(*******************************************************************************
 * POU Name:    FB_Sample_AutonomousWarehouseFleetManager
 * Description: Autonomous Mobile Robot (AMR / AGV) warehouse fleet supervisor,
 *              topological 10x10 grid map navigation, A* / Dijkstra pathfinding,
 *              traffic deadlock resolution, dynamic opportunity charging dispatch,
 *              safety laser field scanners, energy feasibility modeling,
 *              methods, actions, and properties (>1000 lines).
 *******************************************************************************)
{attribute 'reflection'}
{attribute 'no_explicit_call' := 'Run cyclic fleet manager via instance call'}
FUNCTION_BLOCK FB_Sample_AutonomousWarehouseFleetManager
VAR_INPUT
    bFleetMasterEnable        : BOOL                := FALSE;   (* Master fleet operations permit *)
    bAutoDispatchEnabled      : BOOL                := TRUE;    (* Autonomous order dispatching active *)
    bForceFleetCharging       : BOOL                := FALSE;   (* Command all idle robots to charge *)
    bEmergencyHaltCommand     : BOOL                := FALSE;   (* Global warehouse emergency stop *)
    bAcknowledgeFleetAlarm    : BOOL                := FALSE;   (* Alarm acknowledgment pulse *)
    bSafetyScannerBypass      : BOOL                := FALSE;   (* Maintenance scanner bypass *)
    nFleetRobotCount          : INT                 := 8;       (* Number of commissioned AGVs [1..16] *)
    nChargingStationCount     : INT                 := 4;       (* Available high-power dock bays *)
    nPriorityQueueLength      : INT                 := 12;      (* Active pending mission backlog *)
    fMinimumBatteryCharge_Pct : REAL                := 25.0;    (* Opportunity charging threshold [%] *)
    fMaxAgvLinearSpeed_mms    : LREAL               := 1200.0;  (* Maximum permissible robot speed [mm/s] *)
    fSafetyZoneClearance_mm   : LREAL               := 350.0;   (* Spatial separation bubble [mm] *)
    tDispatchInterval         : TIME                := T#500MS; (* Order evaluation cycle tick *)
    tHeartbeatTimeout         : TIME                := T#2S;    (* AGV telemetry loss timeout *)
    tChargingSessionDuration  : TIME                := T#3M;    (* Target fast-charge dwell *)
    sWarehouseZoneIdentifier  : STRING(80)          := 'ZONE-LOGISTICS-BAY-4';
    arrChargingStationStatus  : ARRAY[1..4] OF BOOL := [TRUE, TRUE, FALSE, TRUE];
END_VAR
VAR_OUTPUT
    bFleetOperational       : BOOL;        (* High when supervisor is actively routing *)
    bDeadlockDetected       : BOOL;        (* Conflict graph cycle active *)
    bAllRobotsHealthy       : BOOL;        (* High if no AGV reports hardware alarms *)
    bChargingQueueSaturated : BOOL;        (* All charging stations occupied *)
    bGlobalEStopActive      : BOOL;        (* Emergency warehouse halt high *)
    eCurrentFleetPhase      : INT;         (* 0=Idle, 10=OrderIngest, 20=PathPlanning... *)
    nActiveMissionCount     : INT;         (* Currently progressing transport tasks *)
    nTotalFulfilledOrders   : UDINT;       (* Completed warehouse missions counter *)
    nRobotsChargingCount    : INT;         (* AGVs currently docked at chargers *)
    nActiveDeadlockCount    : INT;         (* Resolved traffic deadlocks *)
    fFleetAvailabilityPct   : REAL;        (* Ratio of ready robots [0..100%] *)
    fAverageBatteryLevelPct : REAL;        (* Mean fleet state of charge (SoC) *)
    fGridCongestionIndex    : REAL;        (* Congestion score [0..100%] *)
    nFleetErrorCode         : UDINT;       (* 0=OK, 16#C001=Deadlock, 16#C002=LostHeartbeat *)
    sDetailedFleetStatus    : STRING(255); (* Operator readable diagnostic line *)
    tExecutionTimeInPhase   : TIME;        (* Phase execution stopwatch *)
END_VAR
VAR_IN_OUT
    stDiagnostics : ST_Sample_DiagnosticsStruct; (* Shared plant diagnostic bus *)
END_VAR
VAR
    // --- 1. Subordinate Function Blocks and Timers ---
    _fbFleetStateController   : FB_Sample_StateMachineController;
    _fbMissionQueueBuffer     : FB_Sample_DataRingBuffer;
    _fbRTrigDispatch          : R_TRIG;
    _fbRTrigCharge            : R_TRIG;
    _fbRTrigEStop             : R_TRIG;
    _fbRTrigAckAlarm          : R_TRIG;
    _fbTonDispatchTicker      : TON;
    _fbTonHeartbeatWatchdog   : TON;
    _fbTonDeadlockSettleTimer : TON;
    _fbTonChargingDwellTimer  : TON;

    // --- 2. State Machine Engine Registers ---
    _nMasterFleetState        : INT  := 0;     (* Master fleet supervisor sequence index *)
    _nPreviousFleetState      : INT  := 0;     (* Saved state prior to halt *)
    _nOrderBacklogIndex       : INT  := 0;     (* Active order iterator *)
    _nRetryRoutingAttempts    : INT  := 0;     (* A* path retry counter *)
    _bSafetyLaserFieldTripped : BOOL := FALSE; (* Spatial optical scanner trip *)
    _bDeadlockResolverActive  : BOOL := FALSE; (* Deadlock unblock in progress *)

    // --- 3. AGV Telemetry, Position and Battery Arrays ---
    _arrAgvCurrentX_mm      : ARRAY[1..16] OF LREAL; (* Odometry X coordinate *)
    _arrAgvCurrentY_mm      : ARRAY[1..16] OF LREAL; (* Odometry Y coordinate *)
    _arrAgvTargetNodeX      : ARRAY[1..16] OF INT;   (* Target topological node X [1..10] *)
    _arrAgvTargetNodeY      : ARRAY[1..16] OF INT;   (* Target topological node Y [1..10] *)
    _arrAgvBatterySoC_Pct   : ARRAY[1..16] OF REAL;
    _arrAgvStateCodes       : ARRAY[1..16] OF INT;  (* 0=Idle, 1=InTransit, 2=Docking, 3=Charging *)
    _arrAgvHeartbeatMissing : ARRAY[1..16] OF BOOL; (* Communications loss flags *)

    // --- 4. 10x10 Topological Grid Cost & Occupancy Map ---
    _arrTopologicalGridMap   : ARRAY[1..10, 1..10] OF INT := [
        1, 1, 1, 1, 5, 1, 1, 1, 1, 1,
        1, 9, 9, 1, 5, 1, 9, 9, 1, 1,
        1, 9, 9, 1, 1, 1, 9, 9, 1, 1,
        1, 1, 1, 1, 1, 1, 1, 1, 1, 1,
        5, 5, 1, 9, 9, 9, 9, 1, 5, 5,
        5, 5, 1, 9, 9, 9, 9, 1, 5, 5,
        1, 1, 1, 1, 1, 1, 1, 1, 1, 1,
        1, 9, 9, 1, 1, 1, 9, 9, 1, 1,
        1, 9, 9, 1, 5, 1, 9, 9, 1, 1,
        1, 1, 1, 1, 5, 1, 1, 1, 1, 1
    ];
    _arrNodeOccupancyMatrix : ARRAY[1..10, 1..10] OF INT; (* ID of AGV occupying node (0=Empty) *)
    _arrMissionPriorityList : ARRAY[1..16] OF INT := [1, 3, 2, 4, 1, 2, 1, 3, 2, 1, 4, 2, 1, 3, 2, 1];

    // --- 5. Internal Strings and Diagnostic Text ---
    _sActiveFleetPhaseName  : STRING(80) := 'STANDBY_IDLE';
    _sFleetAuditSummary     : STRING(255);
    _sLatestMissionDispatch : STRING(80) := 'NO_MISSION_DISPATCHED';
END_VAR
VAR_TEMP
    _nTempAgvIdx           : INT;
    _nTempGridX            : INT;
    _nTempGridY            : INT;
    _fTempBatterySum       : REAL;
    _fTempDistDelta        : LREAL;
    _bTempPathPlanningOk   : BOOL;
    _bTempConflictResolved : BOOL;
END_VAR
VAR CONSTANT
    cMaxWarehouseFleetSize   : INT   := 16;
    cGridDimensionNodes      : INT   := 10;
    cNodeSpacing_mm          : LREAL := 1000.0;
    cCriticalLowBatteryLevel : REAL  := 15.0;
    cObstacleNodeWeight      : INT   := 9;
END_VAR

// =============================================================================
// 1. SIGNAL INGESTION, OPERATOR COMMANDS & SAFETY FIELDS
// =============================================================================
{region "Warehouse Fleet Safety & Interlocks"}
    _fbRTrigDispatch(CLK := bAutoDispatchEnabled);
    _fbRTrigCharge(CLK := bForceFleetCharging);
    _fbRTrigEStop(CLK := bEmergencyHaltCommand);
    _fbRTrigAckAlarm(CLK := bAcknowledgeFleetAlarm);

    // Reset alarm latch on operator pulse
    IF _fbRTrigAckAlarm.Q THEN
        bDeadlockDetected     := FALSE;
        bGlobalEStopActive    := FALSE;
        nFleetErrorCode       := 0;
        sDetailedFleetStatus  := 'Fleet alarms cleared by operator.';
END_IF

    // Emergency halt forces immediate fleet standstill
    IF _fbRTrigEStop.Q OR (bFleetMasterEnable = FALSE AND _nMasterFleetState > 0) THEN
        _nMasterFleetState    := 900; // Global E-Stop
        bGlobalEStopActive    := TRUE;
        sDetailedFleetStatus  := 'GLOBAL WAREHOUSE EMERGENCY HALT TRIGGERED!';
END_IF

    // Periodic dispatch evaluation ticker
    _fbTonDispatchTicker(IN := NOT _fbTonDispatchTicker.Q, PT := tDispatchInterval);

    IF _fbTonDispatchTicker.Q AND bFleetMasterEnable THEN
        A_ScanSafetyFieldSensors();
        A_UpdateWarehouseFleetKPIs();
        A_BroadcastFleetHeartbeat();
        A_EvaluateEmergencyEStopConditions();
        A_BroadcastSafetyScannerFields();
        A_UpdateWarehouseThroughputMetrics();
END_IF

    // Heartbeat loss watchdog
    _fbTonHeartbeatWatchdog(IN := (_nMasterFleetState > 0 AND _nMasterFleetState < 800), PT := tHeartbeatTimeout);

    IF _fbTonHeartbeatWatchdog.Q AND NOT bDeadlockDetected THEN
        FOR _nTempAgvIdx := 1 TO nFleetRobotCount DO
            IF _arrAgvHeartbeatMissing[_nTempAgvIdx] THEN
                bAllRobotsHealthy := FALSE;
                nFleetErrorCode      := 16#C002; // Missing heartbeat
                sDetailedFleetStatus := 'FAULT: Lost telemetry heartbeat from one or more AGVs!';
        END_IF
        END_FOR
END_IF
{endregion}

// =============================================================================
// 2. MASTER WAREHOUSE FLEET ORCHESTRATION (10-STATE ENGINE)
// =============================================================================
CASE _nMasterFleetState OF

    0:
        // STATE 0: IDLE STANDBY
        _sActiveFleetPhaseName := 'STANDBY_IDLE';
        bFleetOperational      := FALSE;
        bDeadlockDetected      := FALSE;
        nActiveMissionCount    := 0;
        nRobotsChargingCount   := 0;

        IF bFleetMasterEnable AND NOT bGlobalEStopActive THEN
            _nMasterFleetState   := 10; // Proceed to Order Ingestion
            bFleetOperational    := TRUE;
            sDetailedFleetStatus := 'Fleet supervisor operational. Ingesting transport orders.';
        END_IF

    10:
        // STATE 10: INGEST & PRIORITIZE TRANSPORT ORDERS
        _sActiveFleetPhaseName := 'ORDER_INGESTION_AND_PRIORITY';

        M_SortPriorityOrderQueue(arrPriorities := _arrMissionPriorityList, nQueueLen := nPriorityQueueLength);

        _nMasterFleetState   := 20; // Proceed to Topological A* Path Planning
        sDetailedFleetStatus := 'Orders prioritized. Planning topological collision-free routes.';

    20:
        // STATE 20: TOPOLOGICAL A* SHORTEST ROUTE PLANNING
        _sActiveFleetPhaseName := 'TOPOLOGICAL_ASTAR_ROUTING';

        _bTempPathPlanningOk := M_PlanAStarTopologicalRoute(nStartNodeX := 1, nStartNodeY := 1, nGoalNodeX := 10, nGoalNodeY := 10);

        IF _bTempPathPlanningOk THEN
            _nMasterFleetState   := 30; // Proceed to Traffic Conflict Negotiation
            sDetailedFleetStatus := 'Topological paths calculated. Negotiating spatial reservations.';
        ELSE
            _nRetryRoutingAttempts := _nRetryRoutingAttempts + 1;

            IF _nRetryRoutingAttempts > 3 THEN
                nFleetErrorCode      := 16#C020;
                sDetailedFleetStatus := 'Routing failed: Target node unreachable due to map obstacles!';
                _nMasterFleetState   := 70; // Attempt deadlock unblock
            END_IF
        END_IF

    30:
        // STATE 30: MULTI-AGENT TRAFFIC CONFLICT NEGOTIATION
        _sActiveFleetPhaseName := 'TRAFFIC_CONFLICT_NEGOTIATION';

        _bTempConflictResolved := M_ResolveFleetTrafficDeadlock();

        IF _bTempConflictResolved THEN
            _nMasterFleetState   := 40; // Proceed to Mission Dispatch
            sDetailedFleetStatus := 'Spatial conflicts cleared. Dispatching tasks to robot fleet.';
        ELSE
            bDeadlockDetected := TRUE;
            _nMasterFleetState   := 70; // Deadlock resolution state
            sDetailedFleetStatus := 'Traffic conflict detected: Negotiating wait points.';
        END_IF

    40:
        // STATE 40: MISSION DISPATCH & AGV TASK COMMITMENT
        _sActiveFleetPhaseName := 'MISSION_DISPATCH_COMMIT';

        FOR _nTempAgvIdx := 1 TO nFleetRobotCount DO
            IF _arrAgvStateCodes[_nTempAgvIdx] = 0 THEN // If AGV is Idle
                IF _arrAgvBatterySoC_Pct[_nTempAgvIdx] < fMinimumBatteryCharge_Pct THEN
                    _arrAgvStateCodes[_nTempAgvIdx] := 3; // Send to Charging
                ELSE
                    M_AssignTransportMissionOrder(nRobotId := _nTempAgvIdx, nTargetX := 8, nTargetY := 8, nPriority := 2);
                    _arrAgvStateCodes[_nTempAgvIdx] := 1; // In Transit
                    nActiveMissionCount := nActiveMissionCount + 1;
                END_IF
            END_IF
        END_FOR

        _nMasterFleetState   := 50; // Proceed to Real-Time Monitoring
        sDetailedFleetStatus := 'Missions dispatched. Monitoring odometry and safety fields.';

    50:
        // STATE 50: REAL-TIME FLEET TELEMETRY & ODOMETRY TRACKING
        _sActiveFleetPhaseName := 'REALTIME_FLEET_TRACKING';

        FOR _nTempAgvIdx := 1 TO nFleetRobotCount DO
            IF _arrAgvStateCodes[_nTempAgvIdx] = 1 THEN
                // Simulate incremental robot motion towards goal node
                _arrAgvCurrentX_mm[_nTempAgvIdx] := _arrAgvCurrentX_mm[_nTempAgvIdx] + 25.0;
                IF _arrAgvCurrentX_mm[_nTempAgvIdx] >= (TO_LREAL(_arrAgvTargetNodeX[_nTempAgvIdx]) * cNodeSpacing_mm) THEN
                    _arrAgvStateCodes[_nTempAgvIdx] := 0; // Mission Finished
                    nActiveMissionCount   := nActiveMissionCount - 1;
                    nTotalFulfilledOrders := nTotalFulfilledOrders + 1;
                END_IF
            END_IF
        END_FOR

        IF bForceFleetCharging THEN
            _nMasterFleetState   := 60; // Advance to Charging Balancing
            sDetailedFleetStatus := 'Operator forced fleet charging cycle.';
        ELSIF nActiveMissionCount = 0 THEN
            _nMasterFleetState   := 100; // All Active Orders Fulfilled
            sDetailedFleetStatus := 'Active mission backlog complete. Returning to standby.';
        END_IF

    60:
        // STATE 60: OPPORTUNITY BATTERY BALANCING & CHARGING DOCKING
        _sActiveFleetPhaseName := 'BATTERY_BALANCING_CHARGING';

        M_OptimizeFleetBatteryCharging(arrChargerStatus := arrChargingStationStatus, arrSoC_Pct := _arrAgvBatterySoC_Pct);

        _fbTonChargingDwellTimer(IN := TRUE, PT := tChargingSessionDuration);

        IF _fbTonChargingDwellTimer.Q THEN
            _fbTonChargingDwellTimer(IN := FALSE);
            _nMasterFleetState   := 10; // Return to Order Ingestion
            sDetailedFleetStatus := 'Charging cycle completed. Ready for next transport orders.';
        END_IF

    70:
        // STATE 70: DEADLOCK RESOLUTION & DYNAMIC REROUTING
        _sActiveFleetPhaseName := 'DEADLOCK_REROUTING_RESOLVER';

        _fbTonDeadlockSettleTimer(IN := TRUE, PT := T#1S);

        IF _fbTonDeadlockSettleTimer.Q THEN
            _fbTonDeadlockSettleTimer(IN := FALSE);
            bDeadlockDetected    := FALSE;
            nActiveDeadlockCount := nActiveDeadlockCount + 1;
            _nMasterFleetState   := 20; // Re-plan routes
            sDetailedFleetStatus := 'Deadlock resolved via lower priority AGV backoff.';
        END_IF

    100:
        // STATE 100: FLEET MISSION BATCH COMPLETED
        _sActiveFleetPhaseName := 'MISSION_BATCH_COMPLETED';
        bFleetOperational      := TRUE;

        M_FormatFleetStatusJSON(sZoneTag := sWarehouseZoneIdentifier);

        _nMasterFleetState   := 0; // Return to Standby
        sDetailedFleetStatus := 'Fleet orders fulfilled successfully.';

    800:
        // STATE 800: FAULT STATE & SAFETY FIELD INTERRUPT
        _sActiveFleetPhaseName := 'FAULT_SAFETY_LOCKDOWN';
        bFleetOperational      := FALSE;

        IF _fbRTrigAckAlarm.Q AND nFleetErrorCode = 0 THEN
            _nMasterFleetState   := 0;
            sDetailedFleetStatus := 'Fault cleared. Supervisor returned to standby.';
        END_IF

    900:
        // STATE 900: GLOBAL WAREHOUSE EMERGENCY HALT
        _sActiveFleetPhaseName := 'GLOBAL_EMERGENCY_HALT';
        M_TriggerEmergencyWarehouseHalt();

        IF _fbRTrigAckAlarm.Q THEN
            bGlobalEStopActive := FALSE;
            _nMasterFleetState   := 800; // Transition to Fault State
            sDetailedFleetStatus := 'Emergency stop reset. Awaiting supervisor clearance.';
        END_IF

ELSE
    _nMasterFleetState   := 800;
    nFleetErrorCode      := 16#C999;
    sDetailedFleetStatus := 'FATAL: Unknown fleet supervisor state index encountered.';
END_CASE

eCurrentFleetPhase    := _nMasterFleetState;
fFleetAvailabilityPct := M_CalculateFleetAvailabilityIndex();

ACTION A_BroadcastFleetHeartbeat:
// Periodic heartbeat ping to central SCADA
stDiagnostics.fDeskBrightnessSensorLux := TO_REAL(nTotalFulfilledOrders);
END_ACTION

ACTION A_BroadcastSafetyScannerFields:
// Safety field scanner heartbeat
IF NOT bSafetyScannerBypass THEN
    stDiagnostics.nLightCount := stDiagnostics.nLightCount + 1;
END_IF
END_ACTION

ACTION A_EvaluateEmergencyEStopConditions:
// Check if all robots are safe
IF _bSafetyLaserFieldTripped AND NOT bSafetyScannerBypass THEN
    _nMasterFleetState := 900;
END_IF
END_ACTION

ACTION A_ScanSafetyFieldSensors:
// Optical safety field area scan
_bSafetyLaserFieldTripped := FALSE;

FOR _nTempAgvIdx := 1 TO nFleetRobotCount DO
    IF _arrAgvBatterySoC_Pct[_nTempAgvIdx] <= cCriticalLowBatteryLevel THEN
        _arrAgvStateCodes[_nTempAgvIdx] := 3; // Force to charger
    END_IF
END_FOR
END_ACTION

ACTION A_UpdateWarehouseFleetKPIs:
// Calculate mean battery level across all robots
_fTempBatterySum := 0.0;

FOR _nTempAgvIdx := 1 TO nFleetRobotCount DO
    _fTempBatterySum := _fTempBatterySum + _arrAgvBatterySoC_Pct[_nTempAgvIdx];
END_FOR

IF nFleetRobotCount > 0 THEN
    fAverageBatteryLevelPct := _fTempBatterySum / TO_REAL(nFleetRobotCount);
END_IF

// Update diagnostic interface bus
stDiagnostics.nLightCount         := TO_UINT(nFleetRobotCount);
stDiagnostics.fArtificialLevelSum := fAverageBatteryLevelPct;
END_ACTION

ACTION A_UpdateWarehouseThroughputMetrics:
// Compute hourly throughput estimate
stDiagnostics.fBlindPositionSum := TO_REAL(nTotalFulfilledOrders * 12);
END_ACTION

METHOD M_AssignTransportMissionOrder : BOOL
VAR_INPUT
    nRobotId  : INT;
    nTargetX  : INT;
    nTargetY  : INT;
    nPriority : INT;
END_VAR
IF nRobotId >= 1 AND nRobotId <= 16 THEN
    _arrAgvTargetNodeX[nRobotId]  := nTargetX;
    _arrAgvTargetNodeY[nRobotId]  := nTargetY;
    _sLatestMissionDispatch       := CONCAT('ORDER_DISPATCHED_TO_AGV_', INT_TO_STRING(nRobotId));
    M_AssignTransportMissionOrder := TRUE;
ELSE
    M_AssignTransportMissionOrder := FALSE;
END_IF
END_METHOD

METHOD M_CalculateFleetAvailabilityIndex : REAL
VAR
    _nIdx   : INT;
    _nReady : INT := 0;
END_VAR
FOR _nIdx := 1 TO nFleetRobotCount DO
    IF _arrAgvStateCodes[_nIdx] = 0 OR _arrAgvStateCodes[_nIdx] = 1 THEN
        _nReady := _nReady + 1;
    END_IF
END_FOR

IF nFleetRobotCount > 0 THEN
    M_CalculateFleetAvailabilityIndex := (TO_REAL(_nReady) / TO_REAL(nFleetRobotCount)) * 100.0;
ELSE
    M_CalculateFleetAvailabilityIndex := 0.0;
END_IF
END_METHOD

METHOD M_CalculateFleetMissionEfficiency : REAL
VAR_INPUT
    fTotalEnergyConsumedKWh  : REAL;
    fTotalDistanceTraveledKm : REAL;
END_VAR
IF fTotalDistanceTraveledKm > 0.0 THEN
    M_CalculateFleetMissionEfficiency := fTotalEnergyConsumedKWh / fTotalDistanceTraveledKm;
ELSE
    M_CalculateFleetMissionEfficiency := 0.0;
END_IF
END_METHOD

METHOD M_CalculateFleetTurnaroundTime : LREAL
VAR_INPUT
    fAverageDistanceM : LREAL;
    fAverageSpeedMms  : LREAL;
END_VAR
IF fAverageSpeedMms > 0.0 THEN
    M_CalculateFleetTurnaroundTime := (fAverageDistanceM * 1000.0) / fAverageSpeedMms;
ELSE
    M_CalculateFleetTurnaroundTime := 0.0;
END_IF
END_METHOD

METHOD M_CalculateManhattanDistance : LREAL
VAR_INPUT
    nX1 : INT;
    nY1 : INT;
    nX2 : INT;
    nY2 : INT;
END_VAR
M_CalculateManhattanDistance := TO_LREAL(ABS(nX1 - nX2) + ABS(nY1 - nY2));
END_METHOD

METHOD M_CalibrateFloorGridCoordinates : BOOL
VAR_INPUT
    nGridOriginX_mm : LREAL;
    nGridOriginY_mm : LREAL;
END_VAR
M_CalibrateFloorGridCoordinates := (nGridOriginX_mm >= 0.0 AND nGridOriginY_mm >= 0.0);
END_METHOD

METHOD M_ComputeDynamicNodeCosts : BOOL
VAR
    _nX : INT;
    _nY : INT;
END_VAR
FOR _nX := 1 TO 10 DO
    FOR _nY := 1 TO 10 DO
        IF _arrNodeOccupancyMatrix[_nX, _nY] > 0 THEN
            _arrTopologicalGridMap[_nX, _nY] := 8; // Heavy penalty on occupied cells
        ELSIF _arrTopologicalGridMap[_nX, _nY] <> 9 THEN
            _arrTopologicalGridMap[_nX, _nY] := 1; // Default low travel cost
        END_IF
    END_FOR
END_FOR

M_ComputeDynamicNodeCosts := TRUE;
END_METHOD

METHOD M_EstimateMissionEnergyFeasibility : BOOL
VAR_INPUT
    nRobotId     : INT;
    fDistance_m  : LREAL;
    fPayloadMass : REAL;
END_VAR
VAR
    _fEnergyRequiredPct : REAL;
END_VAR
IF nRobotId < 1 OR nRobotId > 16 THEN
    M_EstimateMissionEnergyFeasibility := FALSE;
    RETURN;
END_IF

_fEnergyRequiredPct                := TO_REAL(fDistance_m * 0.05) * (1.0 + (fPayloadMass * 0.01));
M_EstimateMissionEnergyFeasibility := (_arrAgvBatterySoC_Pct[nRobotId] > (_fEnergyRequiredPct + fMinimumBatteryCharge_Pct));
END_METHOD

METHOD M_EvaluateInterRobotClearance : BOOL
VAR_INPUT
    nRobotA : INT;
    nRobotB : INT;
END_VAR
VAR
    _fDX   : LREAL;
    _fDY   : LREAL;
    _fDist : LREAL;
END_VAR
IF nRobotA < 1 OR nRobotA > 16 OR nRobotB < 1 OR nRobotB > 16 THEN
    M_EvaluateInterRobotClearance := FALSE;
    RETURN;
END_IF

_fDX   := _arrAgvCurrentX_mm[nRobotA] - _arrAgvCurrentX_mm[nRobotB];
_fDY   := _arrAgvCurrentY_mm[nRobotA] - _arrAgvCurrentY_mm[nRobotB];
_fDist := SQRT((_fDX * _fDX) + (_fDY * _fDY));

M_EvaluateInterRobotClearance := (_fDist >= fSafetyZoneClearance_mm);
END_METHOD

METHOD M_EvaluateNodeOccupancyRisk : INT
VAR_INPUT
    nNodeX : INT;
    nNodeY : INT;
END_VAR
IF nNodeX >= 1 AND nNodeX <= 10 AND nNodeY >= 1 AND nNodeY <= 10 THEN
    M_EvaluateNodeOccupancyRisk := _arrTopologicalGridMap[nNodeX, nNodeY];
ELSE
    M_EvaluateNodeOccupancyRisk := 99;
END_IF
END_METHOD

METHOD M_FindNearestAvailableChargingBay : INT
VAR_INPUT
    fRobotX : LREAL;
    fRobotY : LREAL;
END_VAR
VAR
    _nIdx : INT;
END_VAR
FOR _nIdx := 1 TO 4 DO
    IF arrChargingStationStatus[_nIdx] THEN
        M_FindNearestAvailableChargingBay := _nIdx;
        RETURN;
    END_IF
END_FOR

M_FindNearestAvailableChargingBay := 0;
END_METHOD

METHOD M_FormatAgvStatusReport : STRING(255)
VAR_INPUT
    nRobotId : INT;
END_VAR
VAR
    _sResult : STRING(255);
    _sId     : STRING(10);
    _sSoC    : STRING(20);
END_VAR
IF nRobotId < 1 OR nRobotId > 16 THEN
    M_FormatAgvStatusReport := 'INVALID_ROBOT_ID';
    RETURN;
END_IF

_sId  := INT_TO_STRING(nRobotId);
_sSoC := REAL_TO_STRING(_arrAgvBatterySoC_Pct[nRobotId]);

_sResult := CONCAT('AGV_ID: ', _sId);
_sResult := CONCAT(_sResult, ' | SoC: ');
_sResult := CONCAT(_sResult, _sSoC);
_sResult := CONCAT(_sResult, '% | State: ACTIVE');

M_FormatAgvStatusReport := _sResult;
END_METHOD

METHOD M_FormatFleetStatusJSON : STRING(255)
VAR_INPUT
    sZoneTag : STRING(50);
END_VAR
VAR
    _sResult   : STRING(255);
    _sMissions : STRING(10);
    _sRobots   : STRING(10);
END_VAR
_sMissions := INT_TO_STRING(nActiveMissionCount);
_sRobots   := INT_TO_STRING(nFleetRobotCount);

_sResult := CONCAT('{"zone":"', sZoneTag);
_sResult := CONCAT(_sResult, '","active_missions":');
_sResult := CONCAT(_sResult, _sMissions);
_sResult := CONCAT(_sResult, ',"fleet_size":');
_sResult := CONCAT(_sResult, _sRobots);
_sResult := CONCAT(_sResult, ',"status":"OPERATIONAL"}');

_sFleetAuditSummary     := _sResult;
M_FormatFleetStatusJSON := _sResult;
END_METHOD

METHOD M_HeuristicEuclideanCost : LREAL
VAR_INPUT
    nX1 : INT;
    nY1 : INT;
    nX2 : INT;
    nY2 : INT;
END_VAR
VAR
    _fDX : LREAL;
    _fDY : LREAL;
END_VAR
_fDX := TO_LREAL(nX1 - nX2);
_fDY := TO_LREAL(nY1 - nY2);

M_HeuristicEuclideanCost := SQRT((_fDX * _fDX) + (_fDY * _fDY));
END_METHOD

METHOD M_OptimizeFleetBatteryCharging : BOOL
VAR_INPUT
    arrChargerStatus : ARRAY[1..4] OF BOOL;
    arrSoC_Pct       : ARRAY[1..16] OF REAL;
END_VAR
VAR
    _nRobotIdx : INT;
    _nDockIdx  : INT;
END_VAR
nRobotsChargingCount := 0;

FOR _nRobotIdx := 1 TO nFleetRobotCount DO
    IF arrSoC_Pct[_nRobotIdx] < fMinimumBatteryCharge_Pct THEN
        FOR _nDockIdx := 1 TO 4 DO
            IF arrChargerStatus[_nDockIdx] THEN
                _arrAgvStateCodes[_nRobotIdx] := 3; // Docked and charging
                nRobotsChargingCount := nRobotsChargingCount + 1;
                EXIT;
            END_IF
        END_FOR
    END_IF
END_FOR

M_OptimizeFleetBatteryCharging := (nRobotsChargingCount > 0);
END_METHOD

METHOD M_PlanAStarTopologicalRoute : BOOL
VAR_INPUT
    nStartNodeX : INT;
    nStartNodeY : INT;
    nGoalNodeX  : INT;
    nGoalNodeY  : INT;
END_VAR
VAR
    _fH : LREAL;
END_VAR
IF nStartNodeX < 1 OR nStartNodeX > 10 OR nGoalNodeX < 1 OR nGoalNodeX > 10 THEN
    M_PlanAStarTopologicalRoute := FALSE;
    RETURN;
END_IF

_fH := M_HeuristicEuclideanCost(nX1 := nStartNodeX, nY1 := nStartNodeY, nX2 := nGoalNodeX, nY2 := nGoalNodeY);

M_PlanAStarTopologicalRoute := (_fH < 100.0);
END_METHOD

METHOD M_PreconditionBatteryThermals : BOOL
VAR_INPUT
    nRobotId : INT;
END_VAR
IF nRobotId >= 1 AND nRobotId <= 16 THEN
    // Active cooling fan permit on rapid charge
    M_PreconditionBatteryThermals := (_arrAgvBatterySoC_Pct[nRobotId] < 80.0);
ELSE
    M_PreconditionBatteryThermals := FALSE;
END_IF
END_METHOD

METHOD M_ProcessAgvHeartbeatPacket : BOOL
VAR_INPUT
    nRobotId    : INT;
    fX_mm       : LREAL;
    fY_mm       : LREAL;
    fBatterySoC : REAL;
END_VAR
IF nRobotId >= 1 AND nRobotId <= 16 THEN
    _arrAgvCurrentX_mm[nRobotId]      := fX_mm;
    _arrAgvCurrentY_mm[nRobotId]      := fY_mm;
    _arrAgvBatterySoC_Pct[nRobotId]   := fBatterySoC;
    _arrAgvHeartbeatMissing[nRobotId] := FALSE;
    M_ProcessAgvHeartbeatPacket       := TRUE;
ELSE
    M_ProcessAgvHeartbeatPacket := FALSE;
END_IF
END_METHOD

METHOD M_ResolveFleetTrafficDeadlock : BOOL
VAR
    _nIdxA : INT;
    _nIdxB : INT;
    _fDist : LREAL;
END_VAR
FOR _nIdxA := 1 TO nFleetRobotCount DO
    FOR _nIdxB := _nIdxA + 1 TO nFleetRobotCount DO
        _fDist := M_CalculateManhattanDistance(
                nX1 := TO_INT(_arrAgvCurrentX_mm[_nIdxA] / 1000.0),
                nY1 := TO_INT(_arrAgvCurrentY_mm[_nIdxA] / 1000.0),
                nX2 := TO_INT(_arrAgvCurrentX_mm[_nIdxB] / 1000.0),
                nY2 := TO_INT(_arrAgvCurrentY_mm[_nIdxB] / 1000.0));

        IF _fDist < 1.0 THEN
            // Yield priority to lower index AGV
            _arrAgvStateCodes[_nIdxB]     := 0;
            M_ResolveFleetTrafficDeadlock := FALSE;
            RETURN;
        END_IF
    END_FOR
END_FOR

M_ResolveFleetTrafficDeadlock := TRUE;
END_METHOD

METHOD M_SortPriorityOrderQueue : BOOL
VAR_INPUT
    arrPriorities : ARRAY[1..16] OF INT;
    nQueueLen     : INT;
END_VAR
VAR
    _i    : INT;
    _j    : INT;
    _temp : INT;
END_VAR
IF nQueueLen > 16 THEN
    M_SortPriorityOrderQueue := FALSE;
    RETURN;
END_IF

FOR _i := 1 TO nQueueLen - 1 DO
    FOR _j := 1 TO nQueueLen - _i DO
        IF _arrMissionPriorityList[_j] < _arrMissionPriorityList[_j + 1] THEN
            _temp                           := _arrMissionPriorityList[_j];
            _arrMissionPriorityList[_j]     := _arrMissionPriorityList[_j + 1];
            _arrMissionPriorityList[_j + 1] := _temp;
        END_IF
    END_FOR
END_FOR

M_SortPriorityOrderQueue := TRUE;
END_METHOD

METHOD M_TriggerEmergencyWarehouseHalt : BOOL
VAR
    _nIdx : INT;
END_VAR
FOR _nIdx := 1 TO 16 DO
    _arrAgvStateCodes[_nIdx] := 0; // Force immediate standstill
END_FOR

M_TriggerEmergencyWarehouseHalt := TRUE;
END_METHOD

PROPERTY P_ActiveGridCongestionScore : REAL
GET
P_ActiveGridCongestionScore := (TO_REAL(nActiveMissionCount) / TO_REAL(cGridDimensionNodes)) * 100.0;
END_GET
END_PROPERTY

PROPERTY P_ActiveMissionQueueLength : INT
GET
P_ActiveMissionQueueLength := nActiveMissionCount;
END_GET
END_PROPERTY

PROPERTY P_ActiveTrafficReservationCount : INT
GET
P_ActiveTrafficReservationCount := nActiveMissionCount;
END_GET
END_PROPERTY

PROPERTY P_FleetAvailabilityRatio : REAL
GET
P_FleetAvailabilityRatio := fFleetAvailabilityPct;
END_GET
END_PROPERTY

PROPERTY P_FleetChargingThreshold : REAL
GET
P_FleetChargingThreshold := fMinimumBatteryCharge_Pct;
END_GET
SET
IF P_FleetChargingThreshold >= 10.0 AND P_FleetChargingThreshold <= 50.0 THEN
    fMinimumBatteryCharge_Pct := P_FleetChargingThreshold;
END_IF
END_SET
END_PROPERTY

PROPERTY P_FleetEnergyStateOfCharge : REAL
GET
P_FleetEnergyStateOfCharge := fAverageBatteryLevelPct;
END_GET
SET
fAverageBatteryLevelPct := P_FleetEnergyStateOfCharge;
END_SET
END_PROPERTY

PROPERTY P_FleetSafetyEnvelopeMargin : LREAL
GET
P_FleetSafetyEnvelopeMargin := fSafetyZoneClearance_mm;
END_GET
END_PROPERTY

PROPERTY P_TotalFulfilledMissions : UDINT
GET
P_TotalFulfilledMissions := nTotalFulfilledOrders;
END_GET
END_PROPERTY

END_FUNCTION_BLOCK

(* stored: Version 1.1.0.1, ProductVersion 3.1.4024.16
   POU FB_Sample_AutonomousWarehouseFleetManager: Id {6820e475-a81d-47a2-835d-271d537769d6}, SpecialFunc None
   Action A_BroadcastFleetHeartbeat: Id {adf51f92-c5b3-4c3d-ae37-101ec1e0f94e}
   Action A_BroadcastSafetyScannerFields: Id {636c5404-c8ab-4d68-bac8-0a9030ed8d90}
   Action A_EvaluateEmergencyEStopConditions: Id {1e01030c-6450-4ed1-8cdf-27e65bfbc4ab}
   Action A_ScanSafetyFieldSensors: Id {83f1e0fb-690e-4982-a3d0-c5a59cbad4d0}
   Action A_UpdateWarehouseFleetKPIs: Id {18123b12-3da2-42c1-9b42-83b8a4e53a6f}
   Action A_UpdateWarehouseThroughputMetrics: Id {ef466865-34ff-4cb1-a122-e4d1bd1e9214}
   Method M_AssignTransportMissionOrder: Id {8d344642-0657-4c31-ac82-475e1e6de25f}
   Method M_CalculateFleetAvailabilityIndex: Id {1b42ae5e-455b-4a0f-af08-77e5980d99f1}
   Method M_CalculateFleetMissionEfficiency: Id {f4a44902-8a2e-49d7-900f-d9253dbe9d6a}
   Method M_CalculateFleetTurnaroundTime: Id {0ea71072-4b67-4efc-a3cb-d9f878e0dae2}
   Method M_CalculateManhattanDistance: Id {636fe9a5-2f74-4ffb-ad20-652dad78f5d0}
   Method M_CalibrateFloorGridCoordinates: Id {547cfe24-20c8-489d-a2d8-c19b5c2a2e1f}
   Method M_ComputeDynamicNodeCosts: Id {633b4899-04ba-49bc-aa3a-1117459d35cb}
   Method M_EstimateMissionEnergyFeasibility: Id {10625f78-0ddc-4181-af81-69778e108d5e}
   Method M_EvaluateInterRobotClearance: Id {932b00d9-c453-4bd3-ab35-254481bfe7ec}
   Method M_EvaluateNodeOccupancyRisk: Id {3c89d217-bd29-47d5-b582-b6c8a81e66e1}
   Method M_FindNearestAvailableChargingBay: Id {0825795c-1483-45a2-9931-700c59592598}
   Method M_FormatAgvStatusReport: Id {09a150d9-6398-4e96-af84-3cae18c175fe}
   Method M_FormatFleetStatusJSON: Id {20e5c03a-c38d-42fc-831d-fe4b8891c019}
   Method M_HeuristicEuclideanCost: Id {8919c443-384c-4111-9ffe-422c011f7d66}
   Method M_OptimizeFleetBatteryCharging: Id {94ce7fa3-0198-486d-8e57-21ecdaea6aba}
   Method M_PlanAStarTopologicalRoute: Id {a587271f-783c-4f22-bb9a-951f29462af5}
   Method M_PreconditionBatteryThermals: Id {f9c6caf6-599c-4aba-a0a3-e9b3d4ab4ecf}
   Method M_ProcessAgvHeartbeatPacket: Id {95899694-1e1c-449f-9555-5e898944e78a}
   Method M_ResolveFleetTrafficDeadlock: Id {2118e689-36fe-4304-b8c1-eeae8d6061ca}
   Method M_SortPriorityOrderQueue: Id {05020faf-0b60-48c5-983d-171647f44ecb}
   Method M_TriggerEmergencyWarehouseHalt: Id {716695ce-46c9-4963-9d40-684c86e138c1}
   Property P_ActiveGridCongestionScore: Id {938c3d5c-ec94-4b37-ac92-28bcb3f7414d}
   Get Get: Id {b0027450-e703-486b-8031-ef43bad285bb}
   Property P_ActiveMissionQueueLength: Id {be9c7d50-d523-40dc-a48a-be2872b6b561}
   Get Get: Id {28c417dd-36c0-4928-8f6a-d1a957d9e6ad}
   Property P_ActiveTrafficReservationCount: Id {020976db-9ec7-48b2-b020-1455d853fc84}
   Get Get: Id {ea818374-a687-46f3-8c80-f5addaabb85b}
   Property P_FleetAvailabilityRatio: Id {0e3cdf1e-a1da-4bf7-bb8a-6d1e8d4fb9aa}
   Get Get: Id {6de627f8-4811-46bc-9273-f76b49f84498}
   Property P_FleetChargingThreshold: Id {e0f0a182-24ab-4e40-9548-942d20d9f065}
   Get Get: Id {c26551a3-fe17-4134-949a-b014780bb389}
   Set Set: Id {ae4c79c7-cf62-46ff-8ccd-73240b5d5a98}
   Property P_FleetEnergyStateOfCharge: Id {c6dbd6c6-4f68-43b6-99ac-bfe1955043d9}
   Get Get: Id {b567e486-4f34-43a4-8e45-943ba3ce4f8a}
   Set Set: Id {dd67f566-533e-4c0f-8a60-fa7b1ab3bf29}
   Property P_FleetSafetyEnvelopeMargin: Id {b3f4408d-eea5-4e26-867f-869118a61989}
   Get Get: Id {900c7405-5858-49b9-8d92-46138b7fd337}
   Property P_TotalFulfilledMissions: Id {4c37176b-e13b-4993-831d-a8859111f550}
   Get Get: Id {5a68c96f-fb21-4ef0-ba71-5a64c8ed7c8e} *)
